Staubli VAL3: encodeJState.pgx

public program encodeJState()
  local num l_nRetVal
begin
  // encode prefix length
  l_nRetVal = toBinary(rosJointMsg.prefix.nLength, 1, "-4l", rosJointMsg.prefix.nData)

  // encode header
  l_nRetVal = toBinary(rosJointMsg.header.nMsgType, 1, "-4l", rosJointMsg.header.nData)
  l_nRetVal = toBinary(rosJointMsg.header.nCommType, 1, "-4l", rosJointMsg.header.nData[4])
  l_nRetVal = toBinary(rosJointMsg.header.nReplyCode, 1, "-4l", rosJointMsg.header.nData[8])

  // encode 'sequence' variable of body message (data)
  l_nRetVal = toBinary(rosJointMsg.jointState.nSeq, 1, "-4l", rosJointMsg.body.nData)

  // assuming the remaining elements have zeros assigned by default
  rosJointMsg.jointState.nJoints[0] = jCurrPose.j1 * nDeg2Rad
  rosJointMsg.jointState.nJoints[1] = jCurrPose.j2 * nDeg2Rad
  rosJointMsg.jointState.nJoints[2] = jCurrPose.j3 * nDeg2Rad
  rosJointMsg.jointState.nJoints[3] = jCurrPose.j4 * nDeg2Rad
  rosJointMsg.jointState.nJoints[4] = jCurrPose.j5 * nDeg2Rad
  rosJointMsg.jointState.nJoints[5] = jCurrPose.j6 * nDeg2Rad

  // encode 10 values representing joints[10]
  l_nRetVal = toBinary(rosJointMsg.jointState.nJoints, 10, "4.0l", rosJointMsg.body.nData[4])
end
